// TwinCAT 3 PLC project ph_lv1_io
// Title: tclib_ph_lv1_io
// Company: Poh
// Author: Poh
// ProjectVersion: 0.1.1.0
// ProgramVersion: 3.1.4020.1
// libraries:
//   tclib_ph_lv0, * (Poh)
// project tree:
//   Lv1_IO/Class Interface/ IFC_GENERIC_IO_INTERFACE.TcIO
//   Lv1_IO/Class/ C_GenericDigital_2Channel.TcPOU
// (motion and I/O tree: see PLC project ph_lv0)
// real-time tasks:
//   TASK PlcTask: cycle T#10ms, priority 20, ADS port 350

// ---- Lv1_IO/Class Interface/IFC_GENERIC_IO_INTERFACE.TcIO
INTERFACE IFC_GENERIC_IO_INTERFACE

METHOD IO_Read : RETURN_CODE
VAR_INPUT
	CHANNEL : INT;
	DATA	: POINTER TO LREAL;
END_VAR
END_METHOD

PROPERTY IO_TYPE : INT
GET
END_GET
END_PROPERTY

METHOD IO_Write : RETURN_CODE
VAR_INPUT
	CHANNEL : INT;
	DATA	: LREAL;
END_VAR
END_METHOD

END_INTERFACE

// ---- Lv1_IO/Class/C_GenericDigital_2Channel.TcPOU
FUNCTION_BLOCK C_GenericDigital_2Channel IMPLEMENTS IFC_GENERIC_IO_INTERFACE
VAR_INPUT
END_VAR
VAR_OUTPUT
END_VAR
VAR
	Channel_Data AT %Q* : ARRAY[1..2] OF BOOL;
END_VAR

METHOD IO_Read : ph_lv0.RETURN_CODE
VAR_INPUT
	CHANNEL	: INT;
	DATA	: POINTER TO LREAL;
END_VAR
END_METHOD

{warning 'add property implementation'}
PROPERTY IO_TYPE : INT
GET
END_GET
SET
END_SET
END_PROPERTY

{warning 'add method implementation'}
METHOD IO_Write : ph_lv0.RETURN_CODE
VAR_INPUT
	CHANNEL	: INT;
	DATA	: LREAL;
END_VAR
END_METHOD

END_FUNCTION_BLOCK
